FUNCTION_BLOCK FB_SinGen
VAR_INPUT
	EN :BOOL;
	Offset: LREAL; // where to center the sin wave in the stroke
	Amplitude :LREAL; // how much to multiply the -1 to +1 sin signal by to get the target setpoint
	Reset: BOOL;
	Period : LREAL;
END_VAR
VAR_OUTPUT
	SignalOut :LREAL;
END_VAR
VAR
	TimerPreset: TIME; // freqeuncy of sin depends on this
	K: LREAL;
	N: DINT;
	b_init: BOOL;
	RESULT: LREAL;
	Timer: TON;
	
END_VAR

IF EN THEN
	IF Reset THEN
	b_init := FALSE;
	timer.pt := LREAL_TO_TIME(period);
END_IF

IF NOT b_init THEN
    K :=2*PI/1000; (* DO ONCE *) 
	b_init := TRUE;
END_IF
timer.PT := TimerPreset;
Timer(IN := NOT timer.q);

IF timer.Q AND b_init THEN	// don't step unless initialized
N := N+1; (* REPEAT THIS *)
N :=  N MOD 1000; 
RESULT := SIN(K*N); // feeds out a sin signal from -1 to +1, scale and offset to get appropriate motion profile.
Signalout := ((Result * amplitude) + Global_variables.Position);
END_IF;
ELSE 
	Signalout := 0;
END_IF

END_FUNCTION_BLOCK

(* stored: Version 1.1.0.1, ProductVersion 3.1.4024.4
   POU FB_SinGen: Id {1202d7f5-20e9-4994-b38f-585448299ad7}, SpecialFunc None *)
